FUNCTION F_InLimitTest : BOOL
VAR_INPUT
	fMinimum 	: LREAL;
	fMaximum 	: LREAL;
	fInput 		: LREAL;
END_VAR

//Normal case
// 9 Max
// 5 Test
// 1 Min
IF fMinimum <= fMaximum THEN
	F_InLimitTest := (fInput >= fMinimum) AND (fInput <= fMaximum);
	
//Modulo case	
// 6 | 6  Max
// 5 | 9  Test
// 8 | 8  Min
ELSIF fMinimum > fMaximum THEN
	F_InLimitTest := NOT((fInput > fMaximum) AND (fInput < fMinimum));
END_IF

END_FUNCTION

(* stored: Version 1.1.0.1, ProductVersion 3.1.4024.12
   POU F_InLimitTest: Id {8a35013a-7fd7-4aad-9450-c14e30e8b2f5}, SpecialFunc None *)
